KUKA KRL data list: A15_ljt_global.dat

&ACCESS RV
&COMMENT V_1_4_0
DEFDAT a15_ljt_global PUBLIC
;********************************
;Date: 07.11.2018
;Programmer: AIUT
;Description: Global positions
;********************************




ENDDAT
